Xinje XCPPro project, PLC1: XC2-32 (software 3.3L)

PROGRAM Ladder

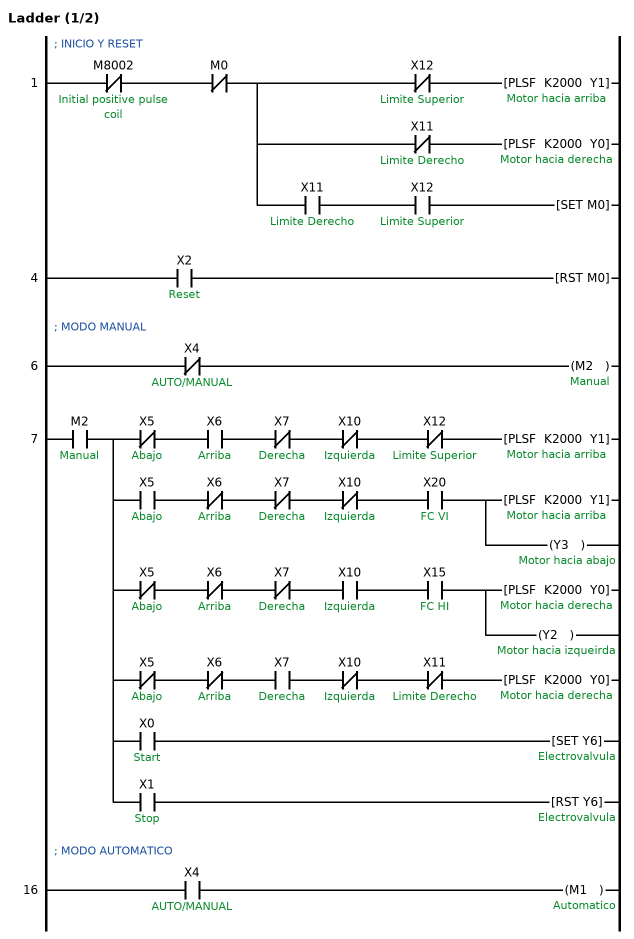
; INICIO Y RESET
LDI    M8002	; Initial positive pulse coil 
ANI    M0
MPS
ANI    X12	; Limite Superior
PLSF   K2000 Y1	; Motor hacia arriba
MRD
ANI    X11	; Limite Derecho
PLSF   K2000 Y0	; Motor hacia derecha
MPP
AND    X11	; Limite Derecho
AND    X12	; Limite Superior
SET    M0
LD     X2	; Reset
RST    M0
; MODO MANUAL
LDI    X4	; AUTO/MANUAL
OUT    M2	; Manual
LD     M2	; Manual
MPS
ANI    X5	; Abajo
AND    X6	; Arriba
ANI    X7	; Derecha
ANI    X10	; Izquierda
ANI    X12	; Limite Superior
PLSF   K2000 Y1	; Motor hacia arriba
MRD
AND    X5	; Abajo
ANI    X6	; Arriba
ANI    X7	; Derecha
ANI    X10	; Izquierda
AND    X20	; FC VI
PLSF   K2000 Y1	; Motor hacia arriba
OUT    Y3	; Motor hacia abajo
MRD
ANI    X5	; Abajo
ANI    X6	; Arriba
ANI    X7	; Derecha
AND    X10	; Izquierda
AND    X15	; FC HI
PLSF   K2000 Y0	; Motor hacia derecha
OUT    Y2	; Motor hacia izqueirda
MRD
ANI    X5	; Abajo
ANI    X6	; Arriba
AND    X7	; Derecha
ANI    X10	; Izquierda
ANI    X11	; Limite Derecho
PLSF   K2000 Y0	; Motor hacia derecha
MRD
AND    X0	; Start
SET    Y6	; Electrovalvula
MPP
AND    X1	; Stop
RST    Y6	; Electrovalvula
; MODO AUTOMATICO
LD     X4	; AUTO/MANUAL
OUT    M1	; Automatico

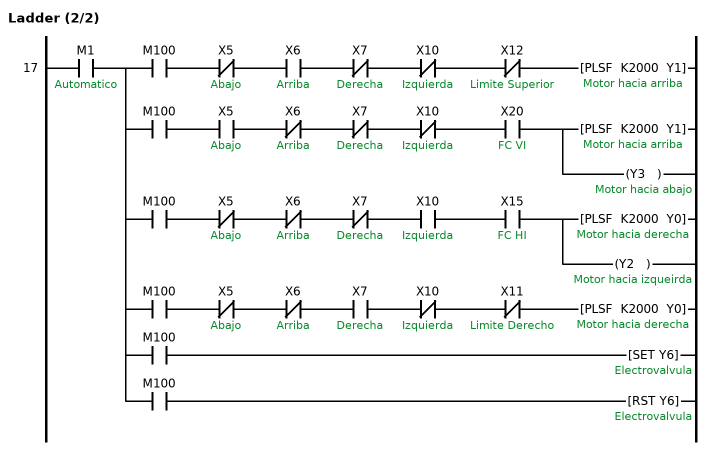
LD     M1	; Automatico
MPS
AND    M100
ANI    X5	; Abajo
AND    X6	; Arriba
ANI    X7	; Derecha
ANI    X10	; Izquierda
ANI    X12	; Limite Superior
PLSF   K2000 Y1	; Motor hacia arriba
MRD
AND    M100
AND    X5	; Abajo
ANI    X6	; Arriba
ANI    X7	; Derecha
ANI    X10	; Izquierda
AND    X20	; FC VI
PLSF   K2000 Y1	; Motor hacia arriba
OUT    Y3	; Motor hacia abajo
MRD
AND    M100
ANI    X5	; Abajo
ANI    X6	; Arriba
ANI    X7	; Derecha
AND    X10	; Izquierda
AND    X15	; FC HI
PLSF   K2000 Y0	; Motor hacia derecha
OUT    Y2	; Motor hacia izqueirda
MRD
AND    M100
ANI    X5	; Abajo
ANI    X6	; Arriba
AND    X7	; Derecha
ANI    X10	; Izquierda
ANI    X11	; Limite Derecho
PLSF   K2000 Y0	; Motor hacia derecha
MRD
AND    M100
SET    Y6	; Electrovalvula
MPP
AND    M100
RST    Y6	; Electrovalvula

COMMENTS (devices not used above)
X3	EMERG
X13	Cilindro Accionado
X14	Cilindro Retraido
X16	FC HD
X17	FC VS
Y4	-
Y5	-
Y7	LEDstart
Y10	LEDstop
Y11	LEDreest